FUNCTION_BLOCK AX_JOB (* Datatyp/Object - Ax Start data *)
VAR_INPUT
//	name						:	STRING(10);
	Fnc														:	INT := 0;
	BufferMode												:	MC_BufferMode := MC_Aborting;(* 	MC_Aborting,
																									MC_Buffered,
																									MC_BlendingLow,
																									MC_BlendingPrevious,
																									MC_BlendingNext,
																									MC_BlendingHigh *)
	Direction												:	MC_Direction := MC_POSITIVE_DIRECTION;	(*	MC_POSITIVE_DIRECTION,
																						   					MC_SHORTeSTATE.WAY,
																						   					MC_NEGATIVE_DIRECTION,
																						   					MC_CURRENT_DIRECTION *)
	Target													:	LREAL	:= 0.0; // target position
	Velo													: 	LREAL	:= 0.0; // target velocity mm/s
	Override												:	LREAL := 100.0; // override
	Acc														:	LREAL := 0.0; // acceleration
	Dec														:	LREAL := 0.0; // deceleration
	Jerk													:	LREAL := 0.0; // jerk
	InTarget												:	BOOL := FALSE;
	InPosWindow												:	BOOL := FALSE;
END_VAR
VAR_OUTPUT
END_VAR
VAR
END_VAR

;

METHOD PUBLIC reset : BOOL
VAR_INPUT
END_VAR
Fnc															:= 0;
BufferMode													:= MC_Aborting;
Direction													:= MC_CURRENT_DIRECTION;
Target														:= 0;
Velo														:= 0;
Override													:= 0;
InTarget													:= FALSE;
InPosWindow													:= FALSE;
reset														:= TRUE;
END_METHOD

END_FUNCTION_BLOCK

(* stored: Version 1.1.0.1, ProductVersion 3.1.4024.3
   POU AX_JOB: Id {9ab18949-101c-4dca-b12d-fe923e02952a}, SpecialFunc None
   Method reset: Id {8c786b13-7b06-4ca9-a464-1ff203e66519} *)
